TYPE ST_GPS_INPUTS :
STRUCT
	x			: LREAL;
END_STRUCT
END_TYPE

(* stored: Version 1.1.0.1, ProductVersion 3.1.4022.11
   DUT ST_GPS_INPUTS: Id {e39b4edf-02d7-4631-851a-b64220d5cdc5} *)
